(*

.. <legal notes>

legal notes
=================
| SPDX-FileCopyrightText: © 2026 Oleksandr Tiutyk <trofimich@gmail.com>
| SPDX-License-Identifier: LGPL-3.0-only
| For details check: LGPL-3.0-only_

.. _LGPL-3.0-only: https://www.gnu.org/licenses/lgpl-3.0.en.html

.. </legal notes>

*)

TYPE ERROR_MESSAGE : WSTRING(2000); END_TYPE

(* stored: Version 1.1.0.1
   DUT ERROR_MESSAGE: Id {72b9ae2b-081e-4ecb-b762-9c7dd5d48450} *)
